// TIA Portal V17 export
// export: Created 2024-09-02T12:50:28.471336Z, ExportSetting WithDefaults, DisplayName Totally Integrated Automation Portal, DisplayVersion V17, DisplayName TIA Portal Openness, DisplayVersion V17, DisplayName TIA Portal Version Control Interface, DisplayVersion V17, DisplayName STEP 7 Professional, DisplayVersion V17, DisplayName STEP 7 Safety, DisplayVersion V17, DisplayName WinCC Professional, DisplayVersion V17
TYPE "TypeSKS_COUNTER"
// stored: IsFailsafeCompliant false
   STRUCT
      "A" : Struct
         CheckStatus : Bool;
         CycleTimeStop : Bool;
         CycleTimeStart : Bool;
         CycleTimeSaving : Bool;
         CycleTimePausePreStp : Bool;
         CycleTimePauseStp : Bool;
         CounterPlusOk : Bool;
         CounterPlusNok : Bool;
      END_STRUCT;
   END_STRUCT;
END_TYPE
